{attribute 'qualified_only'}
{attribute 'strict'}
TYPE E_PalletStopHardwareStates :
(
	Raised,
	Lowered,
	Raising,
	Lowering,
	Fault
);
END_TYPE

(* stored: Version 1.1.0.1, ProductVersion 3.1.4024.12
   DUT E_PalletStopHardwareStates: Id {cc85820b-912c-4f21-8645-1fe6226f0821} *)
